FUNCTION_BLOCK PUBLIC ACMethodDischarging EXTENDS ACMethodRouteBase
VAR_INPUT
END_VAR
VAR_OUTPUT
END_VAR
VAR PERSISTENT
	_Parameter : ACMethodDischargingP;
	_Result : ACMethodDischargingR;
END_VAR

PROPERTY IsValid : BOOL
GET
IsValid := TRUE;
END_GET
END_PROPERTY

PROPERTY Parameter : ACMethodDischargingP
GET
Parameter := _Parameter;
END_GET
SET // PUBLIC
_Parameter := Parameter;
END_SET
END_PROPERTY

PROPERTY Result : ACMethodDischargingR
GET
Result := _Result;
END_GET
SET // PUBLIC
_Result := Result;
END_SET
END_PROPERTY

END_FUNCTION_BLOCK

(* stored: Version 1.1.0.1, ProductVersion 3.1.4022.7
   POU ACMethodDischarging: Id {767368ff-698c-4ac5-8131-bc642d8f48e0}, SpecialFunc None
   Property IsValid: Id {240c4b9b-c94d-424b-8a3b-08228ae6d599}
   Get Get: Id {5162d71e-40bb-41ab-8179-2293debef61b}
   Property Parameter: Id {b09c19ed-611c-4a85-a2a8-8f8377def8ad}
   Get Get: Id {10fbe84c-f830-4dc5-b82f-7bd4dd50bf59}
   Set Set: Id {5980b3ec-cbb4-421c-a04e-92bf6e735dfb}
   Property Result: Id {b59e5876-ddd4-4d25-b14e-58cab793a664}
   Get Get: Id {b58deabd-a5dc-4bc7-a6b9-ecb5bed41c84}
   Set Set: Id {074a6e78-e204-4559-94c0-a1119ece1e63} *)
